// TIA Portal V17 export
// export: Created 2023-03-28T09:21:21.7003707Z, ExportSetting WithDefaults, DisplayName Totally Integrated Automation Portal, DisplayVersion V17 Update 4, DisplayName TIA Portal Openness, DisplayVersion V17 Update 4, DisplayName TIA Portal Version Control Interface, DisplayVersion V17, DisplayName STEP 7 Professional, DisplayVersion V17 Update 4, DisplayName STEP 7 Safety, DisplayVersion V17, DisplayName WinCC Professional, DisplayVersion V17 Update 4
FUNCTION "PCS1 R (PE)" : Void   // FC41, LAD
TITLE = ModBus TCP for PCS Power Electronics
{ S7_Optimized_Access := 'TRUE' }
VERSION : 0.1
// stored: AutoNumber false, IsIECCheckEnabled false, SetENOAutomatically false, UDAEnableTagReadback false
   VAR_TEMP
      rVac : Real;
   END_VAR
   VAR_TEMP   // added for the SCL form of the ladder/FBD networks
      _w1 : Bool;
   END_VAR
BEGIN

REGION Network 1: Function Modbus Client 10ms
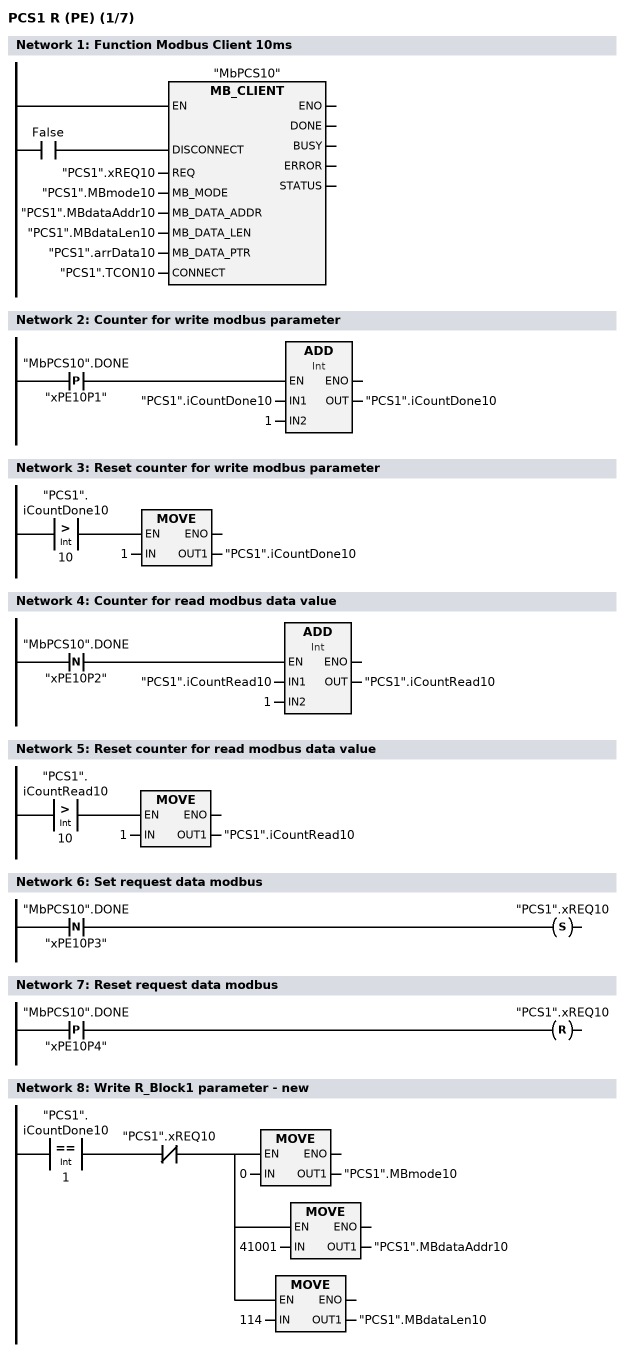
   RUNG wire#powerrail
      "MbPCS10".MB_CLIENT(DISCONNECT := wire#w1, REQ := "PCS1".xREQ10, MB_MODE := "PCS1".MBmode10, MB_DATA_ADDR := "PCS1".MBdataAddr10, MB_DATA_LEN := "PCS1".MBdataLen10, MB_DATA_PTR := "PCS1".arrData10, CONNECT := "PCS1".TCON10, DONE =>, BUSY =>, ERROR =>, STATUS =>)
   END_RUNG
   RUNG wire#powerrail
      Contact( False )
   END_RUNG wire#w1
   // the same network as SCL:
   "MbPCS10"(DISCONNECT := False,   // MB_CLIENT
             REQ := "PCS1".xREQ10,
             MB_MODE := "PCS1".MBmode10,
             MB_DATA_ADDR := "PCS1".MBdataAddr10,
             MB_DATA_LEN := "PCS1".MBdataLen10,
             MB_DATA_PTR := "PCS1".arrData10,
             CONNECT := "PCS1".TCON10);
END_REGION

REGION Network 2: Counter for write modbus parameter
   RUNG wire#powerrail
      P_Contact(operand := "MbPCS10".DONE, bit := "xPE10P1")
      { S7_Templates := "SrcType := Int" } Add(in1 := "PCS1".iCountDone10, in2 := 1, out => "PCS1".iCountDone10)
   END_RUNG
   // the same network as SCL:
   #_w1 := "MbPCS10".DONE AND NOT "xPE10P1";   // rising edge of "MbPCS10".DONE
   "xPE10P1" := "MbPCS10".DONE;
   IF #_w1 THEN "PCS1".iCountDone10 := "PCS1".iCountDone10 + 1; END_IF;
END_REGION

REGION Network 3: Reset counter for write modbus parameter
   RUNG wire#powerrail
      { S7_Templates := "SrcType := Int" } GT_Contact(in1 := "PCS1".iCountDone10, in2 := 10)
      Move(in := 1, out1 => "PCS1".iCountDone10)
   END_RUNG
   // the same network as SCL:
   IF "PCS1".iCountDone10 > 10 THEN "PCS1".iCountDone10 := 1; END_IF;
END_REGION

REGION Network 4: Counter for read modbus data value
   RUNG wire#powerrail
      N_Contact(operand := "MbPCS10".DONE, bit := "xPE10P2")
      { S7_Templates := "SrcType := Int" } Add(in1 := "PCS1".iCountRead10, in2 := 1, out => "PCS1".iCountRead10)
   END_RUNG
   // the same network as SCL:
   #_w1 := NOT "MbPCS10".DONE AND "xPE10P2";   // falling edge of "MbPCS10".DONE
   "xPE10P2" := "MbPCS10".DONE;
   IF #_w1 THEN "PCS1".iCountRead10 := "PCS1".iCountRead10 + 1; END_IF;
END_REGION

REGION Network 5: Reset counter for read modbus data value
   RUNG wire#powerrail
      { S7_Templates := "SrcType := Int" } GT_Contact(in1 := "PCS1".iCountRead10, in2 := 10)
      Move(in := 1, out1 => "PCS1".iCountRead10)
   END_RUNG
   // the same network as SCL:
   IF "PCS1".iCountRead10 > 10 THEN "PCS1".iCountRead10 := 1; END_IF;
END_REGION

REGION Network 6: Set request data modbus
   RUNG wire#powerrail
      N_Contact(operand := "MbPCS10".DONE, bit := "xPE10P3")
      S_Coil( "PCS1".xREQ10 )
   END_RUNG
   // the same network as SCL:
   #_w1 := NOT "MbPCS10".DONE AND "xPE10P3";   // falling edge of "MbPCS10".DONE
   "xPE10P3" := "MbPCS10".DONE;
   IF #_w1 THEN "PCS1".xREQ10 := TRUE; END_IF;
END_REGION

REGION Network 7: Reset request data modbus
   RUNG wire#powerrail
      P_Contact(operand := "MbPCS10".DONE, bit := "xPE10P4")
      R_Coil( "PCS1".xREQ10 )
   END_RUNG
   // the same network as SCL:
   #_w1 := "MbPCS10".DONE AND NOT "xPE10P4";   // rising edge of "MbPCS10".DONE
   "xPE10P4" := "MbPCS10".DONE;
   IF #_w1 THEN "PCS1".xREQ10 := FALSE; END_IF;
END_REGION

REGION Network 8: Write R_Block1 parameter - new
   RUNG wire#powerrail
      { S7_Templates := "SrcType := Int" } EQ_Contact(in1 := "PCS1".iCountDone10, in2 := 1)
      I_Contact( "PCS1".xREQ10 )
      wire#w1
      Move(in := 0, out1 => "PCS1".MBmode10)
   END_RUNG
   RUNG wire#w1
      Move(in := 41001, out1 => "PCS1".MBdataAddr10)
   END_RUNG
   RUNG wire#w1
      Move(in := 114, out1 => "PCS1".MBdataLen10)
   END_RUNG
   // the same network as SCL:
   IF ("PCS1".iCountDone10 = 1) AND NOT "PCS1".xREQ10 THEN
       "PCS1".MBmode10 := 0;
       "PCS1".MBdataAddr10 := 41001;
       "PCS1".MBdataLen10 := 114;
   END_IF;
END_REGION

REGION Network 9: Read R_Block1 data value - new
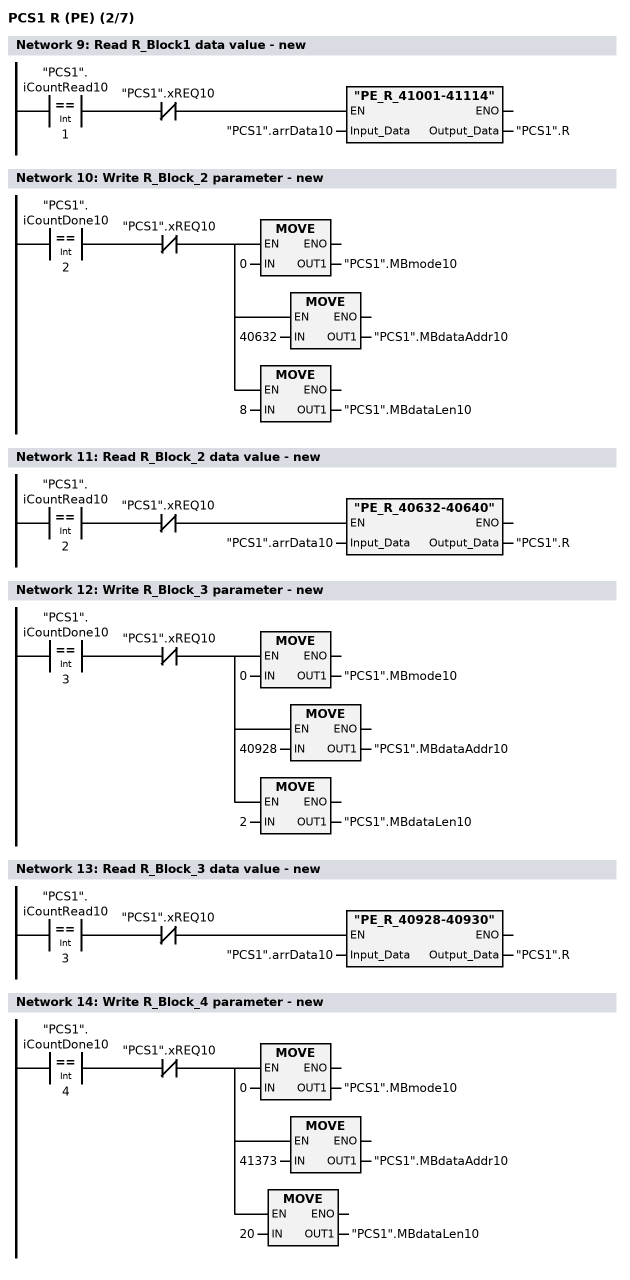
   RUNG wire#powerrail
      { S7_Templates := "SrcType := Int" } EQ_Contact(in1 := "PCS1".iCountRead10, in2 := 1)
      I_Contact( "PCS1".xREQ10 )
      "PE_R_41001-41114"(Input_Data := "PCS1".arrData10, Output_Data => "PCS1".R)
   END_RUNG
   // the same network as SCL:
   IF ("PCS1".iCountRead10 = 1) AND NOT "PCS1".xREQ10 THEN
       "PE_R_41001-41114"(Input_Data := "PCS1".arrData10, Output_Data => "PCS1".R);
   END_IF;
END_REGION

REGION Network 10: Write R_Block_2 parameter - new
   RUNG wire#powerrail
      { S7_Templates := "SrcType := Int" } EQ_Contact(in1 := "PCS1".iCountDone10, in2 := 2)
      I_Contact( "PCS1".xREQ10 )
      wire#w1
      Move(in := 0, out1 => "PCS1".MBmode10)
   END_RUNG
   RUNG wire#w1
      Move(in := 40632, out1 => "PCS1".MBdataAddr10)
   END_RUNG
   RUNG wire#w1
      Move(in := 8, out1 => "PCS1".MBdataLen10)
   END_RUNG
   // the same network as SCL:
   IF ("PCS1".iCountDone10 = 2) AND NOT "PCS1".xREQ10 THEN
       "PCS1".MBmode10 := 0;
       "PCS1".MBdataAddr10 := 40632;
       "PCS1".MBdataLen10 := 8;
   END_IF;
END_REGION

REGION Network 11: Read R_Block_2 data value - new
   RUNG wire#powerrail
      { S7_Templates := "SrcType := Int" } EQ_Contact(in1 := "PCS1".iCountRead10, in2 := 2)
      I_Contact( "PCS1".xREQ10 )
      "PE_R_40632-40640"(Input_Data := "PCS1".arrData10, Output_Data => "PCS1".R)
   END_RUNG
   // the same network as SCL:
   IF ("PCS1".iCountRead10 = 2) AND NOT "PCS1".xREQ10 THEN
       "PE_R_40632-40640"(Input_Data := "PCS1".arrData10, Output_Data => "PCS1".R);
   END_IF;
END_REGION

REGION Network 12: Write R_Block_3 parameter - new
   RUNG wire#powerrail
      { S7_Templates := "SrcType := Int" } EQ_Contact(in1 := "PCS1".iCountDone10, in2 := 3)
      I_Contact( "PCS1".xREQ10 )
      wire#w1
      Move(in := 0, out1 => "PCS1".MBmode10)
   END_RUNG
   RUNG wire#w1
      Move(in := 40928, out1 => "PCS1".MBdataAddr10)
   END_RUNG
   RUNG wire#w1
      Move(in := 2, out1 => "PCS1".MBdataLen10)
   END_RUNG
   // the same network as SCL:
   IF ("PCS1".iCountDone10 = 3) AND NOT "PCS1".xREQ10 THEN
       "PCS1".MBmode10 := 0;
       "PCS1".MBdataAddr10 := 40928;
       "PCS1".MBdataLen10 := 2;
   END_IF;
END_REGION

REGION Network 13: Read R_Block_3 data value - new
   RUNG wire#powerrail
      { S7_Templates := "SrcType := Int" } EQ_Contact(in1 := "PCS1".iCountRead10, in2 := 3)
      I_Contact( "PCS1".xREQ10 )
      "PE_R_40928-40930"(Input_Data := "PCS1".arrData10, Output_Data => "PCS1".R)
   END_RUNG
   // the same network as SCL:
   IF ("PCS1".iCountRead10 = 3) AND NOT "PCS1".xREQ10 THEN
       "PE_R_40928-40930"(Input_Data := "PCS1".arrData10, Output_Data => "PCS1".R);
   END_IF;
END_REGION

REGION Network 14: Write R_Block_4 parameter - new
   RUNG wire#powerrail
      { S7_Templates := "SrcType := Int" } EQ_Contact(in1 := "PCS1".iCountDone10, in2 := 4)
      I_Contact( "PCS1".xREQ10 )
      wire#w1
      Move(in := 0, out1 => "PCS1".MBmode10)
   END_RUNG
   RUNG wire#w1
      Move(in := 41373, out1 => "PCS1".MBdataAddr10)
   END_RUNG
   RUNG wire#w1
      Move(in := 20, out1 => "PCS1".MBdataLen10)
   END_RUNG
   // the same network as SCL:
   IF ("PCS1".iCountDone10 = 4) AND NOT "PCS1".xREQ10 THEN
       "PCS1".MBmode10 := 0;
       "PCS1".MBdataAddr10 := 41373;
       "PCS1".MBdataLen10 := 20;
   END_IF;
END_REGION

REGION Network 15: Read R_Block_4 data value - new
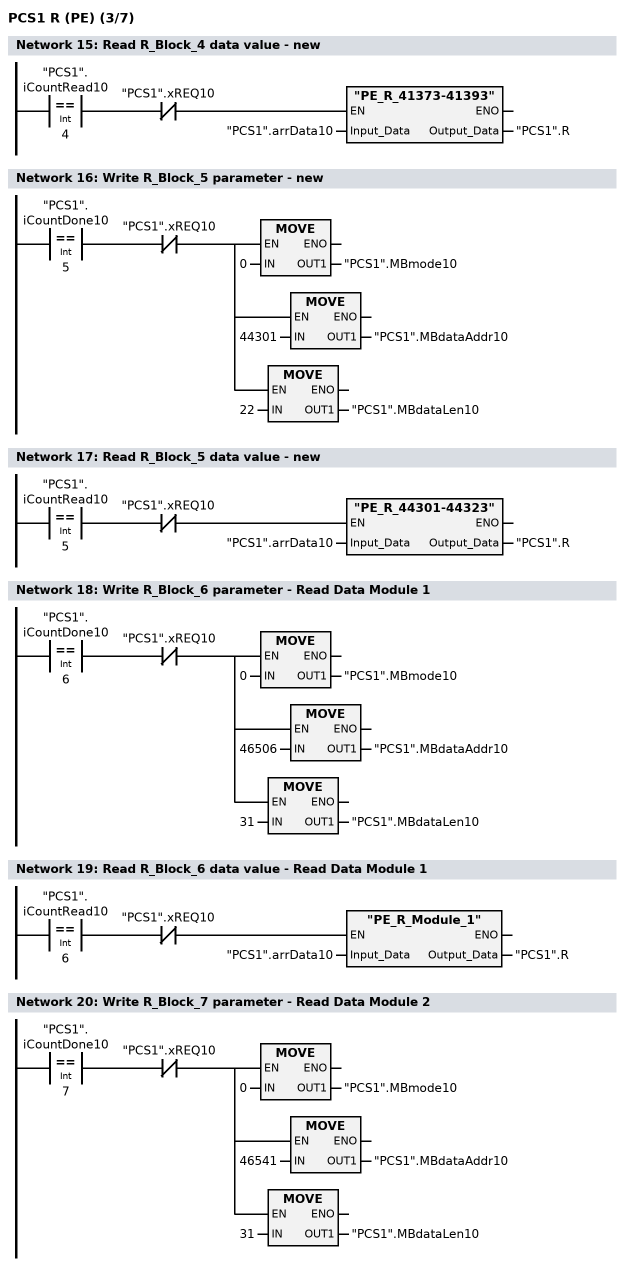
   RUNG wire#powerrail
      { S7_Templates := "SrcType := Int" } EQ_Contact(in1 := "PCS1".iCountRead10, in2 := 4)
      I_Contact( "PCS1".xREQ10 )
      "PE_R_41373-41393"(Input_Data := "PCS1".arrData10, Output_Data => "PCS1".R)
   END_RUNG
   // the same network as SCL:
   IF ("PCS1".iCountRead10 = 4) AND NOT "PCS1".xREQ10 THEN
       "PE_R_41373-41393"(Input_Data := "PCS1".arrData10, Output_Data => "PCS1".R);
   END_IF;
END_REGION

REGION Network 16: Write R_Block_5 parameter - new
   RUNG wire#powerrail
      { S7_Templates := "SrcType := Int" } EQ_Contact(in1 := "PCS1".iCountDone10, in2 := 5)
      I_Contact( "PCS1".xREQ10 )
      wire#w1
      Move(in := 0, out1 => "PCS1".MBmode10)
   END_RUNG
   RUNG wire#w1
      Move(in := 44301, out1 => "PCS1".MBdataAddr10)
   END_RUNG
   RUNG wire#w1
      Move(in := 22, out1 => "PCS1".MBdataLen10)
   END_RUNG
   // the same network as SCL:
   IF ("PCS1".iCountDone10 = 5) AND NOT "PCS1".xREQ10 THEN
       "PCS1".MBmode10 := 0;
       "PCS1".MBdataAddr10 := 44301;
       "PCS1".MBdataLen10 := 22;
   END_IF;
END_REGION

REGION Network 17: Read R_Block_5 data value - new
   RUNG wire#powerrail
      { S7_Templates := "SrcType := Int" } EQ_Contact(in1 := "PCS1".iCountRead10, in2 := 5)
      I_Contact( "PCS1".xREQ10 )
      "PE_R_44301-44323"(Input_Data := "PCS1".arrData10, Output_Data => "PCS1".R)
   END_RUNG
   // the same network as SCL:
   IF ("PCS1".iCountRead10 = 5) AND NOT "PCS1".xREQ10 THEN
       "PE_R_44301-44323"(Input_Data := "PCS1".arrData10, Output_Data => "PCS1".R);
   END_IF;
END_REGION

REGION Network 18: Write R_Block_6 parameter - Read Data Module 1
   RUNG wire#powerrail
      { S7_Templates := "SrcType := Int" } EQ_Contact(in1 := "PCS1".iCountDone10, in2 := 6)
      I_Contact( "PCS1".xREQ10 )
      wire#w1
      Move(in := 0, out1 => "PCS1".MBmode10)
   END_RUNG
   RUNG wire#w1
      Move(in := 46506, out1 => "PCS1".MBdataAddr10)
   END_RUNG
   RUNG wire#w1
      Move(in := 31, out1 => "PCS1".MBdataLen10)
   END_RUNG
   // the same network as SCL:
   IF ("PCS1".iCountDone10 = 6) AND NOT "PCS1".xREQ10 THEN
       "PCS1".MBmode10 := 0;
       "PCS1".MBdataAddr10 := 46506;
       "PCS1".MBdataLen10 := 31;
   END_IF;
END_REGION

REGION Network 19: Read R_Block_6 data value - Read Data Module 1
   RUNG wire#powerrail
      { S7_Templates := "SrcType := Int" } EQ_Contact(in1 := "PCS1".iCountRead10, in2 := 6)
      I_Contact( "PCS1".xREQ10 )
      "PE_R_Module_1"(Input_Data := "PCS1".arrData10, Output_Data => "PCS1".R)
   END_RUNG
   // the same network as SCL:
   IF ("PCS1".iCountRead10 = 6) AND NOT "PCS1".xREQ10 THEN
       "PE_R_Module_1"(Input_Data := "PCS1".arrData10, Output_Data => "PCS1".R);
   END_IF;
END_REGION

REGION Network 20: Write R_Block_7 parameter - Read Data Module 2
   RUNG wire#powerrail
      { S7_Templates := "SrcType := Int" } EQ_Contact(in1 := "PCS1".iCountDone10, in2 := 7)
      I_Contact( "PCS1".xREQ10 )
      wire#w1
      Move(in := 0, out1 => "PCS1".MBmode10)
   END_RUNG
   RUNG wire#w1
      Move(in := 46541, out1 => "PCS1".MBdataAddr10)
   END_RUNG
   RUNG wire#w1
      Move(in := 31, out1 => "PCS1".MBdataLen10)
   END_RUNG
   // the same network as SCL:
   IF ("PCS1".iCountDone10 = 7) AND NOT "PCS1".xREQ10 THEN
       "PCS1".MBmode10 := 0;
       "PCS1".MBdataAddr10 := 46541;
       "PCS1".MBdataLen10 := 31;
   END_IF;
END_REGION

REGION Network 21: Read R_Block_7 data value - Read Data Module 2
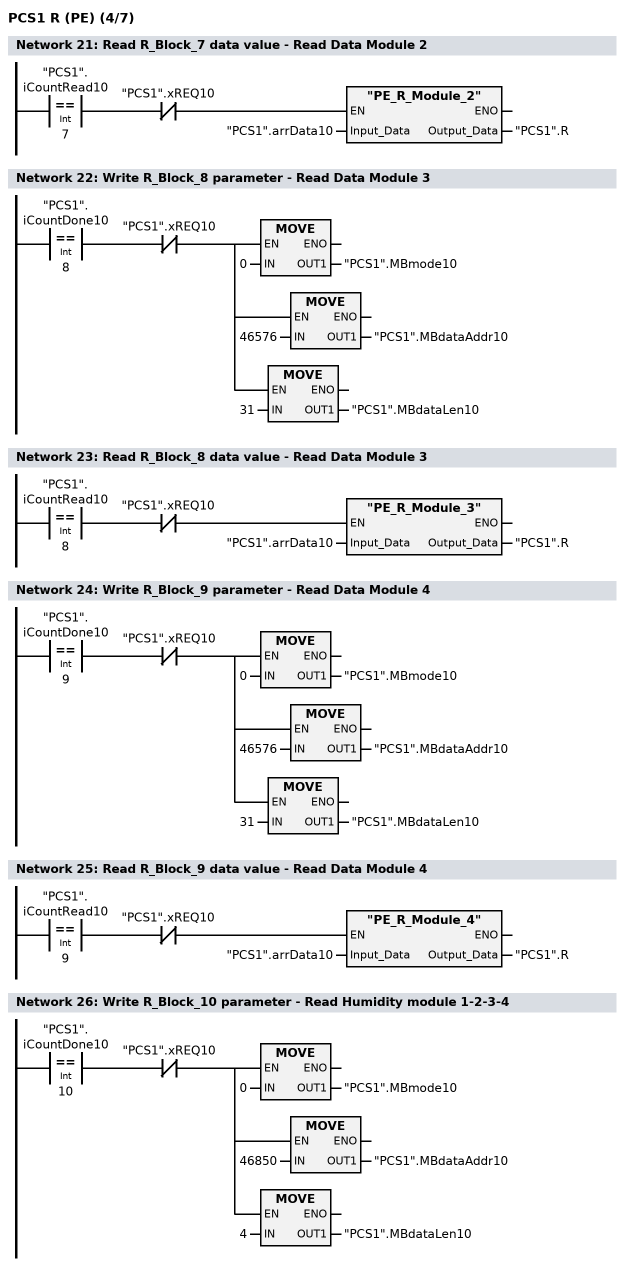
   RUNG wire#powerrail
      { S7_Templates := "SrcType := Int" } EQ_Contact(in1 := "PCS1".iCountRead10, in2 := 7)
      I_Contact( "PCS1".xREQ10 )
      "PE_R_Module_2"(Input_Data := "PCS1".arrData10, Output_Data => "PCS1".R)
   END_RUNG
   // the same network as SCL:
   IF ("PCS1".iCountRead10 = 7) AND NOT "PCS1".xREQ10 THEN
       "PE_R_Module_2"(Input_Data := "PCS1".arrData10, Output_Data => "PCS1".R);
   END_IF;
END_REGION

REGION Network 22: Write R_Block_8 parameter - Read Data Module 3
   RUNG wire#powerrail
      { S7_Templates := "SrcType := Int" } EQ_Contact(in1 := "PCS1".iCountDone10, in2 := 8)
      I_Contact( "PCS1".xREQ10 )
      wire#w1
      Move(in := 0, out1 => "PCS1".MBmode10)
   END_RUNG
   RUNG wire#w1
      Move(in := 46576, out1 => "PCS1".MBdataAddr10)
   END_RUNG
   RUNG wire#w1
      Move(in := 31, out1 => "PCS1".MBdataLen10)
   END_RUNG
   // the same network as SCL:
   IF ("PCS1".iCountDone10 = 8) AND NOT "PCS1".xREQ10 THEN
       "PCS1".MBmode10 := 0;
       "PCS1".MBdataAddr10 := 46576;
       "PCS1".MBdataLen10 := 31;
   END_IF;
END_REGION

REGION Network 23: Read R_Block_8 data value - Read Data Module 3
   RUNG wire#powerrail
      { S7_Templates := "SrcType := Int" } EQ_Contact(in1 := "PCS1".iCountRead10, in2 := 8)
      I_Contact( "PCS1".xREQ10 )
      "PE_R_Module_3"(Input_Data := "PCS1".arrData10, Output_Data => "PCS1".R)
   END_RUNG
   // the same network as SCL:
   IF ("PCS1".iCountRead10 = 8) AND NOT "PCS1".xREQ10 THEN
       "PE_R_Module_3"(Input_Data := "PCS1".arrData10, Output_Data => "PCS1".R);
   END_IF;
END_REGION

REGION Network 24: Write R_Block_9 parameter - Read Data Module 4
   RUNG wire#powerrail
      { S7_Templates := "SrcType := Int" } EQ_Contact(in1 := "PCS1".iCountDone10, in2 := 9)
      I_Contact( "PCS1".xREQ10 )
      wire#w1
      Move(in := 0, out1 => "PCS1".MBmode10)
   END_RUNG
   RUNG wire#w1
      Move(in := 46576, out1 => "PCS1".MBdataAddr10)
   END_RUNG
   RUNG wire#w1
      Move(in := 31, out1 => "PCS1".MBdataLen10)
   END_RUNG
   // the same network as SCL:
   IF ("PCS1".iCountDone10 = 9) AND NOT "PCS1".xREQ10 THEN
       "PCS1".MBmode10 := 0;
       "PCS1".MBdataAddr10 := 46576;
       "PCS1".MBdataLen10 := 31;
   END_IF;
END_REGION

REGION Network 25: Read R_Block_9 data value - Read Data Module 4
   RUNG wire#powerrail
      { S7_Templates := "SrcType := Int" } EQ_Contact(in1 := "PCS1".iCountRead10, in2 := 9)
      I_Contact( "PCS1".xREQ10 )
      "PE_R_Module_4"(Input_Data := "PCS1".arrData10, Output_Data => "PCS1".R)
   END_RUNG
   // the same network as SCL:
   IF ("PCS1".iCountRead10 = 9) AND NOT "PCS1".xREQ10 THEN
       "PE_R_Module_4"(Input_Data := "PCS1".arrData10, Output_Data => "PCS1".R);
   END_IF;
END_REGION

REGION Network 26: Write R_Block_10 parameter - Read Humidity module 1-2-3-4
   RUNG wire#powerrail
      { S7_Templates := "SrcType := Int" } EQ_Contact(in1 := "PCS1".iCountDone10, in2 := 10)
      I_Contact( "PCS1".xREQ10 )
      wire#w1
      Move(in := 0, out1 => "PCS1".MBmode10)
   END_RUNG
   RUNG wire#w1
      Move(in := 46850, out1 => "PCS1".MBdataAddr10)
   END_RUNG
   RUNG wire#w1
      Move(in := 4, out1 => "PCS1".MBdataLen10)
   END_RUNG
   // the same network as SCL:
   IF ("PCS1".iCountDone10 = 10) AND NOT "PCS1".xREQ10 THEN
       "PCS1".MBmode10 := 0;
       "PCS1".MBdataAddr10 := 46850;
       "PCS1".MBdataLen10 := 4;
   END_IF;
END_REGION

REGION Network 27: Read R_Block_10 data value - Read Humidity module 1-2-3-4
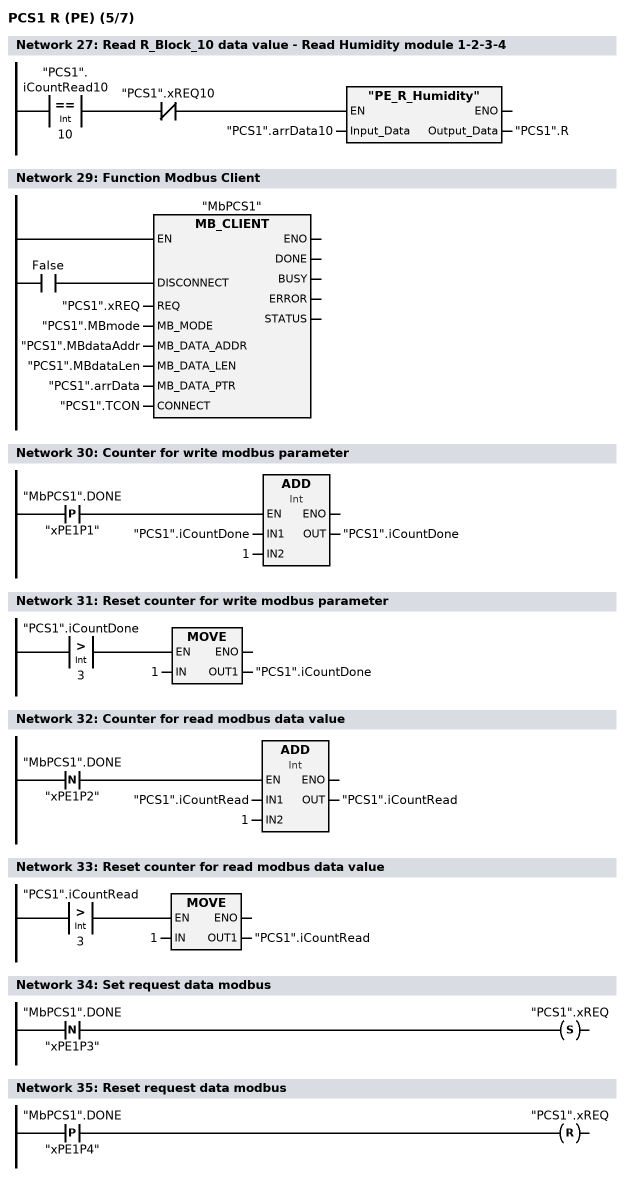
   RUNG wire#powerrail
      { S7_Templates := "SrcType := Int" } EQ_Contact(in1 := "PCS1".iCountRead10, in2 := 10)
      I_Contact( "PCS1".xREQ10 )
      "PE_R_Humidity"(Input_Data := "PCS1".arrData10, Output_Data => "PCS1".R)
   END_RUNG
   // the same network as SCL:
   IF ("PCS1".iCountRead10 = 10) AND NOT "PCS1".xREQ10 THEN
       "PE_R_Humidity"(Input_Data := "PCS1".arrData10, Output_Data => "PCS1".R);
   END_IF;
END_REGION

REGION Network 29: Function Modbus Client
   RUNG wire#powerrail
      "MbPCS1".MB_CLIENT(DISCONNECT := wire#w1, REQ := "PCS1".xREQ, MB_MODE := "PCS1".MBmode, MB_DATA_ADDR := "PCS1".MBdataAddr, MB_DATA_LEN := "PCS1".MBdataLen, MB_DATA_PTR := "PCS1".arrData, CONNECT := "PCS1".TCON, DONE =>, BUSY =>, ERROR =>, STATUS =>)
   END_RUNG
   RUNG wire#powerrail
      Contact( False )
   END_RUNG wire#w1
   // the same network as SCL:
   "MbPCS1"(DISCONNECT := False,   // MB_CLIENT
            REQ := "PCS1".xREQ,
            MB_MODE := "PCS1".MBmode,
            MB_DATA_ADDR := "PCS1".MBdataAddr,
            MB_DATA_LEN := "PCS1".MBdataLen,
            MB_DATA_PTR := "PCS1".arrData,
            CONNECT := "PCS1".TCON);
END_REGION

REGION Network 30: Counter for write modbus parameter
   RUNG wire#powerrail
      P_Contact(operand := "MbPCS1".DONE, bit := "xPE1P1")
      { S7_Templates := "SrcType := Int" } Add(in1 := "PCS1".iCountDone, in2 := 1, out => "PCS1".iCountDone)
   END_RUNG
   // the same network as SCL:
   #_w1 := "MbPCS1".DONE AND NOT "xPE1P1";   // rising edge of "MbPCS1".DONE
   "xPE1P1" := "MbPCS1".DONE;
   IF #_w1 THEN "PCS1".iCountDone := "PCS1".iCountDone + 1; END_IF;
END_REGION

REGION Network 31: Reset counter for write modbus parameter
   RUNG wire#powerrail
      { S7_Templates := "SrcType := Int" } GT_Contact(in1 := "PCS1".iCountDone, in2 := 3)
      Move(in := 1, out1 => "PCS1".iCountDone)
   END_RUNG
   // the same network as SCL:
   IF "PCS1".iCountDone > 3 THEN "PCS1".iCountDone := 1; END_IF;
END_REGION

REGION Network 32: Counter for read modbus data value
   RUNG wire#powerrail
      N_Contact(operand := "MbPCS1".DONE, bit := "xPE1P2")
      { S7_Templates := "SrcType := Int" } Add(in1 := "PCS1".iCountRead, in2 := 1, out => "PCS1".iCountRead)
   END_RUNG
   // the same network as SCL:
   #_w1 := NOT "MbPCS1".DONE AND "xPE1P2";   // falling edge of "MbPCS1".DONE
   "xPE1P2" := "MbPCS1".DONE;
   IF #_w1 THEN "PCS1".iCountRead := "PCS1".iCountRead + 1; END_IF;
END_REGION

REGION Network 33: Reset counter for read modbus data value
   RUNG wire#powerrail
      { S7_Templates := "SrcType := Int" } GT_Contact(in1 := "PCS1".iCountRead, in2 := 3)
      Move(in := 1, out1 => "PCS1".iCountRead)
   END_RUNG
   // the same network as SCL:
   IF "PCS1".iCountRead > 3 THEN "PCS1".iCountRead := 1; END_IF;
END_REGION

REGION Network 34: Set request data modbus
   RUNG wire#powerrail
      N_Contact(operand := "MbPCS1".DONE, bit := "xPE1P3")
      S_Coil( "PCS1".xREQ )
   END_RUNG
   // the same network as SCL:
   #_w1 := NOT "MbPCS1".DONE AND "xPE1P3";   // falling edge of "MbPCS1".DONE
   "xPE1P3" := "MbPCS1".DONE;
   IF #_w1 THEN "PCS1".xREQ := TRUE; END_IF;
END_REGION

REGION Network 35: Reset request data modbus
   RUNG wire#powerrail
      P_Contact(operand := "MbPCS1".DONE, bit := "xPE1P4")
      R_Coil( "PCS1".xREQ )
   END_RUNG
   // the same network as SCL:
   #_w1 := "MbPCS1".DONE AND NOT "xPE1P4";   // rising edge of "MbPCS1".DONE
   "xPE1P4" := "MbPCS1".DONE;
   IF #_w1 THEN "PCS1".xREQ := FALSE; END_IF;
END_REGION

REGION Network 37: Write RW_Block1 parameter - da controllare password
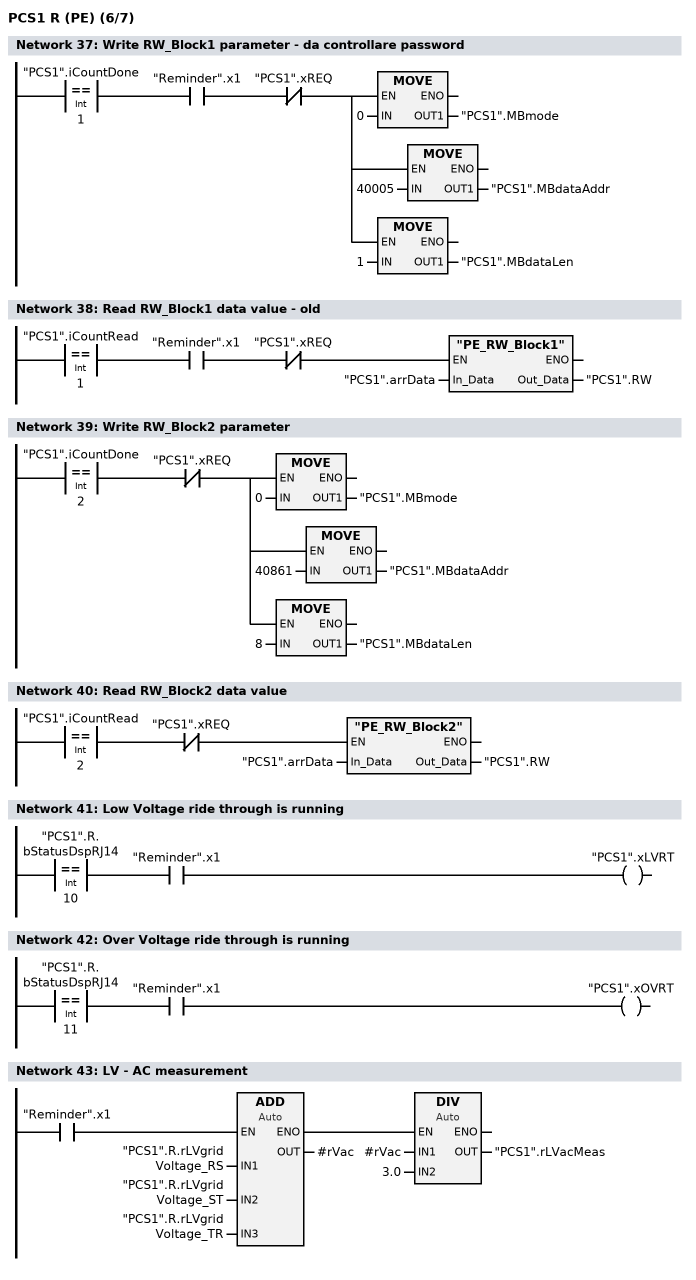
   RUNG wire#powerrail
      { S7_Templates := "SrcType := Int" } EQ_Contact(in1 := "PCS1".iCountDone, in2 := 1)
      Contact( "Reminder".x1 )
      I_Contact( "PCS1".xREQ )
      wire#w1
      Move(in := 0, out1 => "PCS1".MBmode)
   END_RUNG
   RUNG wire#w1
      Move(in := 40005, out1 => "PCS1".MBdataAddr)
   END_RUNG
   RUNG wire#w1
      Move(in := 1, out1 => "PCS1".MBdataLen)
   END_RUNG
   // the same network as SCL:
   IF ("PCS1".iCountDone = 1) AND "Reminder".x1 AND NOT "PCS1".xREQ THEN
       "PCS1".MBmode := 0;
       "PCS1".MBdataAddr := 40005;
       "PCS1".MBdataLen := 1;
   END_IF;
END_REGION

REGION Network 38: Read RW_Block1 data value - old
   RUNG wire#powerrail
      { S7_Templates := "SrcType := Int" } EQ_Contact(in1 := "PCS1".iCountRead, in2 := 1)
      Contact( "Reminder".x1 )
      I_Contact( "PCS1".xREQ )
      "PE_RW_Block1"(In_Data := "PCS1".arrData, Out_Data => "PCS1".RW)
   END_RUNG
   // the same network as SCL:
   IF ("PCS1".iCountRead = 1) AND "Reminder".x1 AND NOT "PCS1".xREQ THEN
       "PE_RW_Block1"(In_Data := "PCS1".arrData, Out_Data => "PCS1".RW);
   END_IF;
END_REGION

REGION Network 39: Write RW_Block2 parameter
   RUNG wire#powerrail
      { S7_Templates := "SrcType := Int" } EQ_Contact(in1 := "PCS1".iCountDone, in2 := 2)
      I_Contact( "PCS1".xREQ )
      wire#w1
      Move(in := 0, out1 => "PCS1".MBmode)
   END_RUNG
   RUNG wire#w1
      Move(in := 40861, out1 => "PCS1".MBdataAddr)
   END_RUNG
   RUNG wire#w1
      Move(in := 8, out1 => "PCS1".MBdataLen)
   END_RUNG
   // the same network as SCL:
   IF ("PCS1".iCountDone = 2) AND NOT "PCS1".xREQ THEN
       "PCS1".MBmode := 0;
       "PCS1".MBdataAddr := 40861;
       "PCS1".MBdataLen := 8;
   END_IF;
END_REGION

REGION Network 40: Read RW_Block2 data value
   RUNG wire#powerrail
      { S7_Templates := "SrcType := Int" } EQ_Contact(in1 := "PCS1".iCountRead, in2 := 2)
      I_Contact( "PCS1".xREQ )
      "PE_RW_Block2"(In_Data := "PCS1".arrData, Out_Data => "PCS1".RW)
   END_RUNG
   // the same network as SCL:
   IF ("PCS1".iCountRead = 2) AND NOT "PCS1".xREQ THEN
       "PE_RW_Block2"(In_Data := "PCS1".arrData, Out_Data => "PCS1".RW);
   END_IF;
END_REGION

REGION Network 41: Low Voltage ride through is running
   RUNG wire#powerrail
      { S7_Templates := "SrcType := Int" } EQ_Contact(in1 := "PCS1".R.bStatusDspRJ14, in2 := 10)
      Contact( "Reminder".x1 )
      Coil( "PCS1".xLVRT )
   END_RUNG
   // the same network as SCL:
   "PCS1".xLVRT := ("PCS1".R.bStatusDspRJ14 = 10) AND "Reminder".x1;
END_REGION

REGION Network 42: Over Voltage ride through is running
   RUNG wire#powerrail
      { S7_Templates := "SrcType := Int" } EQ_Contact(in1 := "PCS1".R.bStatusDspRJ14, in2 := 11)
      Contact( "Reminder".x1 )
      Coil( "PCS1".xOVRT )
   END_RUNG
   // the same network as SCL:
   "PCS1".xOVRT := ("PCS1".R.bStatusDspRJ14 = 11) AND "Reminder".x1;
END_REGION

REGION Network 43: LV - AC measurement
   RUNG wire#powerrail
      Contact( "Reminder".x1 )
      Add(in1 := "PCS1".R.rLVgridVoltage_RS, in2 := "PCS1".R.rLVgridVoltage_ST, in3 := "PCS1".R.rLVgridVoltage_TR, out => #rVac)
      Div(in1 := #rVac, in2 := 3.0, out => "PCS1".rLVacMeas)
   END_RUNG
   // the same network as SCL:
   IF "Reminder".x1 THEN
       #rVac := "PCS1".R.rLVgridVoltage_RS + "PCS1".R.rLVgridVoltage_ST + "PCS1".R.rLVgridVoltage_TR;
       "PCS1".rLVacMeas := #rVac / 3.0;
   END_IF;
END_REGION

REGION Network 44: MV - AC measurement
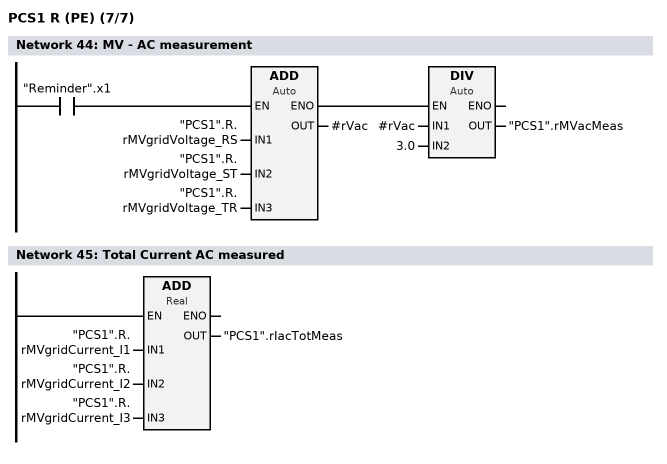
   RUNG wire#powerrail
      Contact( "Reminder".x1 )
      Add(in1 := "PCS1".R.rMVgridVoltage_RS, in2 := "PCS1".R.rMVgridVoltage_ST, in3 := "PCS1".R.rMVgridVoltage_TR, out => #rVac)
      Div(in1 := #rVac, in2 := 3.0, out => "PCS1".rMVacMeas)
   END_RUNG
   // the same network as SCL:
   IF "Reminder".x1 THEN
       #rVac := "PCS1".R.rMVgridVoltage_RS + "PCS1".R.rMVgridVoltage_ST + "PCS1".R.rMVgridVoltage_TR;
       "PCS1".rMVacMeas := #rVac / 3.0;
   END_IF;
END_REGION

REGION Network 45: Total Current AC measured
   RUNG wire#powerrail
      { S7_Templates := "SrcType := Real" } Add(in1 := "PCS1".R.rMVgridCurrent_I1, in2 := "PCS1".R.rMVgridCurrent_I2, in3 := "PCS1".R.rMVgridCurrent_I3, out => "PCS1".rIacTotMeas)
   END_RUNG
   // the same network as SCL:
   "PCS1".rIacTotMeas := "PCS1".R.rMVgridCurrent_I1 + "PCS1".R.rMVgridCurrent_I2 + "PCS1".R.rMVgridCurrent_I3;
END_REGION
END_FUNCTION
